FUNCTION_BLOCK FB_ShippingTransCV_LeftSide EXTENDS FB_ActionBasic
VAR_INPUT
    xExecute    : BOOL;
    xAbort      : BOOL;
	xReset		: BOOL;
	TimeOut  	: LREAL := 60; // Unit : s
    Cylinder 	: REFERENCE TO UNI_CylinderList;
	Motor		: REFERENCE TO UNI_MotorList;
	Input		: REFERENCE TO ST_InputTable;
	OutPut		: REFERENCE TO ST_OutputTable;
	ShippingTransCVRequest_LeftSide : BOOL;
	RobotStatus	: ST_StatusBasic;		// robot Service 
END_VAR
VAR_OUTPUT
	xAborted : BOOL;
    iErrorID : INT;
    ErrorMsg : STRING;
END_VAR
VAR
	// model setting 
	StateBehaviour   : CBML.ETrigATo;
    CurrentPosition : ST_PositionTable;
	fbExecuteEdgeDetect :FB_EdgeDetect;
	Reset_Rtrig 	:R_TRIG;
	uiCyclicStep    : UINT := 0;
	
	//Timer
	TON_DelayArrivedDetect	: TON;
	TON_TransCVAllowDelay	: TON;
END_VAR

THIS^.IBehaviourModel := StateBehaviour;

StateBehaviour(xExecute := xExecute,
              xAbort := xAbort OR fbExecuteEdgeDetect.xFallingEdge,
              udiTimeOut := LREAL_TO_UDINT( TimeOut*1000000),
              xDone => xDone,
              xBusy => xBusy,
              xError => xError,
              xAborted => xAborted);
			  
//Make sure that C# turns off execute to shut down the service
fbExecuteEdgeDetect(xInput :=xExecute);
  
//Error Msg
iErrorID := StateBehaviour._model.iErrorID;
ErrorMsg := M_GetErrorMsg(xErrorID := iErrorID);

//Reset
Reset_Rtrig(CLK:= xReset);
IF Reset_Rtrig.Q THEN
	StateBehaviour.ResetModel(xCommit:=xReset);
END_IF

//Action
A00_BaseUnit();

ACTION A00_BaseUnit:
TON_DelayArrivedDetect(PT:=T#1S);
TON_TransCVAllowDelay(PT :=T#1S);
END_ACTION

METHOD CleanupAction
VAR_INPUT
    xAbortProposed : BOOL;
    iErrorIDProposed: INT;
END_VAR
VAR_OUTPUT
    xComplete : BOOL := TRUE;
    xAbort: BOOL := xAbortProposed;
 	iErrorID : INT := iErrorIDProposed;
END_VAR
END_METHOD

METHOD CyclicAction
VAR_INPUT
    itfTimingController : CBML.ITimingController;
END_VAR
VAR_OUTPUT
    xComplete : BOOL := TRUE;
    iErrorID : INT := 0;
END_VAR
xComplete := FALSE;


CASE uiCyclicStep OF 
	0:	// robot status , send allow signal
		IF ShippingTransCVRequest_LeftSide AND NOT RobotStatus.Busy THEN
			TON_TransCVAllowDelay.IN := TRUE;
			OutPut.bShippingTransCV_Leftside_Allow := TRUE;
		END_IF
		IF TON_TransCVAllowDelay.Q THEN
			OutPut.bShippingTransCV_Leftside_Allow := FALSE;
			uiCyclicStep := 100;
		END_IF

	100:	//check HansLaser cancel signal
		TON_TransCVAllowDelay.IN := FALSE;
		IF NOT Input.bShippingTransCV_Leftside_Arrived THEN 
			xComplete := TRUE;
		END_IF
END_CASE

IF Input.bHansLaserMachineError THEN
	iErrorID := 10;
END_IF
END_METHOD

METHOD ExitAction
VAR_INPUT
    xAfterCleanup : BOOL;
    xInCopyCode : BOOL;
END_VAR
END_METHOD

METHOD M_GetErrorMsg : T_MaxString
VAR_INPUT
	xErrorID: INT;
END_VAR

VAR
	
END_VAR
CASE xErrorID OF
	0:
		M_GetErrorMsg := 'No Error';
	1:
		M_GetErrorMsg := 'FB_ShippingTransCV_LeftSide ErrorID 1: Action time out';
///
	10:
		M_GetErrorMsg := 'FB_ShippingTransCV_LeftSide ErrorID 10: HansLaser Machine Error';
	11:
		M_GetErrorMsg := 'FB_ShippingTransCV_LeftSide ErrorID 11: Wrong Command , TransCV not IntargetPosition';
END_CASE
END_METHOD

METHOD ResetAction
VAR_OUTPUT
    xComplete : BOOL := TRUE;
END_VAR
xComplete := FALSE;

ShippingTransCVRequest_LeftSide 		:= FALSE;
OutPut.bShippingTransCV_Leftside_Allow := FALSE;

TON_DelayArrivedDetect.IN := FALSE;
TON_TransCVAllowDelay.IN := FALSE;

uiCyclicStep := 0;

xComplete := TRUE;
END_METHOD

METHOD StartAction
VAR_OUTPUT
    xComplete : BOOL := TRUE;
	iErrorID : INT := 0;
END_VAR
xComplete := FALSE;

ShippingTransCVRequest_LeftSide 		:= FALSE;
OutPut.bShippingTransCV_Leftside_Allow := FALSE;

uiCyclicStep := 0;

TON_DelayArrivedDetect.IN := FALSE;
TON_TransCVAllowDelay.IN := FALSE;


xComplete := TRUE;

IF Input.bHansLaserMachineError THEN
	iErrorID := 10;
END_IF

IF NOT Input.bShippingTransCV_Leftside_Arrived THEN
	iErrorID := 11;
END_IF
END_METHOD

END_FUNCTION_BLOCK

(* stored: Version 1.1.0.1, ProductVersion 3.1.4024.13
   POU FB_ShippingTransCV_LeftSide: Id {3251d885-8122-4d6b-97be-a737c3f81fdd}, SpecialFunc None
   Folder Action: Id {bb766b2f-628b-4e49-b30f-ceca13d5809f}
   Action A00_BaseUnit: Id {34085937-00e1-496c-b8a9-c92e8ffa9d5e}
   Method CleanupAction: Id {78be9580-f971-4554-9741-9b798826f82a}
   Method CyclicAction: Id {8c013b82-1618-4b69-a150-95cdf7f2f1c3}
   Method ExitAction: Id {23b115d1-7595-4767-94b4-e4093c085e87}
   Method M_GetErrorMsg: Id {d9ab3778-f06d-470b-a3b8-c7cceef991fe}
   Method ResetAction: Id {f31d21b4-d912-43b2-bc88-5832af690956}
   Method StartAction: Id {8d70a5a7-c8e7-4c6f-9470-f1ae13f3fd85} *)
